Fanuc KAREL source: kt00473.KL

-- PROVISIONAL review KL for V940-1; original PC SHA256 0371eafa9219509a9e9cca941041106151adcfc5f26eb9b1abc420b263c957c6
-- Incomplete behavior may be omitted. Consult companion uncertainty JSON. Do not deploy.
PROGRAM KT00473
%NOLOCKGROUP
VAR
  OUT : BOOLEAN
-- UNRESOLVED_DECL P1 type=000101
-- UNRESOLVED_DECL P2 type=000101
BEGIN
  -- V9_ZERO_TABLE_METADATA_HINT layout=0001; no indexed target words; source/name/runtime held
  -- UNRESOLVED_PC offsets 5-28; opcodes 49,49,AC,23
  -- UNRESOLVED_PC offsets 33-37; opcodes 7F
END KT00473
